(* PLC project , Arduino SRL Arduino PLC IDE Application 1.0.3.1 *)
(* stored: companyURL https://www.axelsoftware.it/, creationDateTime 2023-12-08T15:45:33 *)

VAR_GLOBAL  (* Global_vars *)
  cnt : INT;
  pickSeq : BOOL := FALSE;
  curSeq : INT := 10;
  auto : BOOL;
  manMode : BOOL;
  pickIndex : INT := 0;
  placePositionsY : ARRAY[0..3] OF INT := [7200, 10200, 13650, 16650];
  placeIndex : INT;
  placeSeq : BOOL;
  laserSeq : INT;
  pickPositionX : INT := 7975;
  placeClearZ : INT := 13600;
  workDone : BOOL := FALSE;
  pushSeq : BOOL;
  cutPositionsY : ARRAY[0..9] OF INT := [20970, 19000, 17030, 15060, 13090, 11120, 9150, 7180, 5210, 3240];
  cutBackX : INT := 15600;
  cutFrontX : INT := 18500;
  cutSeq : BOOL := FALSE;
  moveSpeed : INT := 375;
  min0 : INT := 0;
  min1 : INT := 0;
  hour0 : INT := 0;
  hour1 : INT := 0;
  placedCur : ARRAY[0..3] OF INT;
  timeReal : ARRAY[0..3] OF INT;
  timeRTC : ARRAY[0..3] OF INT;
  Solenoids AT %MX3.2 : ARRAY[0..3] OF BOOL;
  cutDigit : INT;
  engraveSeq : BOOL;
END_VAR

VAR_GLOBAL CONSTANT  (* Global_vars_Constant *)
  ZTop : INT := 14800;
  XOFF : INT := 0;
  YOFF : INT := 0;
  ZOFF : INT := 0;
  pickPositionsY : ARRAY[0..9] OF INT := [20900, 18930, 16960, 14990, 13020, 11050, 9080, 7100, 5140, 3600];
  pickClearanceZ : INT := 10000;
  placePositionX : INT := 19400;
  PBTimeOff : INT := 200;
  pushClearanceX : INT := 16350;
END_VAR

VAR_GLOBAL  (* I_O_mappings_DIO *)
  Sol1 AT %MX3.2 : BOOL;
  Sol2 AT %MX3.3 : BOOL;
  Sol3 AT %MX3.4 : BOOL;
  EnableXYZ AT %MX3.0 : BOOL;
  EnableA AT %MX3.1 : BOOL;
  Sol4 AT %MX3.5 : BOOL;
END_VAR

VAR_GLOBAL  (* I_O_mappings_DI *)
  XHome AT %IX0.0 : BOOL;
  YHome AT %IX0.1 : BOOL;
  ZHome AT %IX0.2 : BOOL;
END_VAR

VAR_GLOBAL  (* I_O_mappings_DO *)
  home2 : BOOL;
END_VAR

VAR_GLOBAL  (* I_O_mappings_AO *)
  laserPWM AT %QD1.1 : REAL;
END_VAR

PROGRAM TimeGetter

timeRTC[0] := minute MOD 10;
timeRTC[1] := minute / 10;

timeRTC[2] := hour MOD 10;
timeRTC[3] := hour / 10;

/* placedCur[3] is hour1 and also most significant.
If time changes, reset placedCur[x] to -1 and drop piece. */
IF(placedCur[3] = -1) THEN
	placeIndex := 3;

ELSIF(placedCur[2] = -1) THEN
	placeIndex := 2;

ELSIF(placedCur[1] = -1) THEN
	placeIndex := 1;
	
ELSIF(placedCur[0] = -1) THEN
	placeIndex := 0;

END_IF;

//set placedCur[x] to -1 when time changes, and not in motion.
END_PROGRAM

FUNCTION_BLOCK Engrave0
  VAR_INPUT
    YPOS0 : INT;
    XPOS0 : INT;
    XPOSACT : INT;
    YPOSACT : INT;
  END_VAR
  VAR_OUTPUT
    LASERPWM : REAL;
    XPOSOUT : INT;
    YPOSOUT : INT;
  END_VAR
  VAR_EXTERNAL
    curSeq : INT;
  END_VAR

IF (curSeq = 20) THEN
XPOSOUT := XPOS0 + 450;
YPOSOUT := YPOS0 + 450;
END_IF;


//Fire laser while moving through sequence
IF (curSeq > 20) AND (curSeq < 100) THEN
LASERPWM := 0.8;
ELSE
LASERPWM := 0.0;
END_IF;

IF (curSeq = 21) THEN
XPOSOUT := XPOS0 + 2505;
YPOSOUT := YPOS0 + 450;
END_IF;

IF (curSeq = 22) THEN
XPOSOUT := XPOS0 + 2505;
YPOSOUT := YPOS0 + 1520;
END_IF;

IF (curSeq = 23) THEN
XPOSOUT := XPOS0 + 450;
YPOSOUT := YPOS0 + 1520;
END_IF;

IF (curSeq = 24) THEN
XPOSOUT := XPOS0 + 450;
YPOSOUT := YPOS0 + 550;
END_IF;



//Move to next sequence if current sequence reaches its requested position.
//Might need another condition so CURSEQ doesn't keep incrementing
IF (XPOSOUT = XPOSACT) AND (YPOSOUT = YPOSACT) THEN 
curSeq := curSeq + 1;
END_IF;


//End of engrave sequence looking for 100
//23 is a placeholder for last sequence
IF(curSeq > 24) THEN
curSeq := 100;
LASERPWM := 0.0;

END_IF;
END_FUNCTION_BLOCK

FUNCTION_BLOCK Engrave1
  VAR_INPUT
    YPOS0 : INT;
    XPOS0 : INT;
    XPOSACT : INT;
    YPOSACT : INT;
  END_VAR
  VAR_OUTPUT
    LASERPWM : REAL;
    XPOSOUT : INT;
    YPOSOUT : INT;
  END_VAR
  VAR_EXTERNAL
    curSeq : INT;
  END_VAR

IF (curSeq = 20) THEN
XPOSOUT := XPOS0 + 768;
YPOSOUT := YPOS0 + 1303;
END_IF;


//Fire laser while moving through sequence
IF (curSeq > 20) AND (curSeq < 100) THEN
LASERPWM := 0.8;
ELSE
LASERPWM := 0.0;
END_IF;

IF (curSeq = 21) THEN
XPOSOUT := XPOS0 + 450;
YPOSOUT := YPOS0 + 985;
END_IF;

IF (curSeq = 22) THEN
XPOSOUT := XPOS0 + 2405;
YPOSOUT := YPOS0 + 985;
END_IF;

IF (curSeq = 23) THEN
XPOSOUT := XPOS0 + 2405;
YPOSOUT := YPOS0 + 1520;
END_IF;

IF (curSeq = 24) THEN
XPOSOUT := XPOS0 + 2505;
YPOSOUT := YPOS0 + 1520;
END_IF;

IF (curSeq = 25) THEN
XPOSOUT := XPOS0 + 2505;
YPOSOUT := YPOS0 + 450;
END_IF;



//Move to next sequence if current sequence reaches its requested position.
//Might need another condition so CURSEQ doesn't keep incrementing
IF (XPOSOUT = XPOSACT) AND (YPOSOUT = YPOSACT) THEN
curSeq := curSeq + 1;
END_IF;


//End of engrave sequence looking for 100
//23 is a placeholder for last sequence
IF(curSeq > 25) THEN
curSeq := 100;
LASERPWM := 0.0;
END_IF;
END_FUNCTION_BLOCK

FUNCTION_BLOCK Engrave2
  VAR_INPUT
    YPOS0 : INT;
    XPOS0 : INT;
    XPOSACT : INT;
    YPOSACT : INT;
  END_VAR
  VAR_OUTPUT
    LASERPWM : REAL;
    XPOSOUT : INT;
    YPOSOUT : INT;
  END_VAR
  VAR_EXTERNAL
    curSeq : INT;
  END_VAR

IF (curSeq = 20) THEN
XPOSOUT := XPOS0 + 900;
YPOSOUT := YPOS0 + 1520;
END_IF;


//Fire laser while moving through sequence
IF (curSeq > 20) AND (curSeq < 100) THEN
LASERPWM := 0.8;
ELSE
LASERPWM := 0.0;
END_IF;

IF (curSeq = 21) THEN
XPOSOUT := XPOS0 + 450;
YPOSOUT := YPOS0 + 1520;
END_IF;

IF (curSeq = 22) THEN
XPOSOUT := XPOS0 + 450;
YPOSOUT := YPOS0 + 450;
END_IF;

IF (curSeq = 23) THEN
XPOSOUT := XPOS0 + 1480;
YPOSOUT := YPOS0 + 450;
END_IF;

IF (curSeq = 24) THEN
XPOSOUT := XPOS0 + 1480;
YPOSOUT := YPOS0 + 1520;
END_IF;

IF (curSeq = 25) THEN
XPOSOUT := XPOS0 + 2505;
YPOSOUT := YPOS0 + 1520;
END_IF;

IF (curSeq = 26) THEN
XPOSOUT := XPOS0 + 2505;
YPOSOUT := YPOS0 + 450;
END_IF;



//Move to next sequence if current sequence reaches its requested position.
//Might need another condition so CURSEQ doesn't keep incrementing
IF (XPOSOUT = XPOSACT) AND (YPOSOUT = YPOSACT) THEN
curSeq := curSeq + 1;
END_IF;


//End of engrave sequence looking for 100
//23 is a placeholder for last sequence
IF(curSeq > 26) THEN
curSeq := 100;
LASERPWM := 0.0;
END_IF;
END_FUNCTION_BLOCK

FUNCTION_BLOCK Engrave3
  VAR_INPUT
    YPOS0 : INT;
    XPOS0 : INT;
    XPOSACT : INT;
    YPOSACT : INT;
  END_VAR
  VAR_OUTPUT
    LASERPWM : REAL;
    XPOSOUT : INT;
    YPOSOUT : INT;
  END_VAR
  VAR_EXTERNAL
    curSeq : INT;
  END_VAR

IF (curSeq = 20) THEN
XPOSOUT := XPOS0 + 450;
YPOSOUT := YPOS0 + 1520;
END_IF;


//Fire laser while moving through sequence
IF (curSeq > 20) AND (curSeq < 100) THEN
LASERPWM := 0.8;
ELSE
LASERPWM := 0.0;
END_IF;

IF (curSeq = 21) THEN
XPOSOUT := XPOS0 + 450;
YPOSOUT := YPOS0 + 450;
END_IF;

IF (curSeq = 22) THEN
XPOSOUT := XPOS0 + 1475;
YPOSOUT := YPOS0 + 450;
END_IF;

IF (curSeq = 23) THEN
XPOSOUT := XPOS0 + 1475;
YPOSOUT := YPOS0 + 1520;
END_IF;

IF (curSeq = 24) THEN
XPOSOUT := XPOS0 + 1575;
YPOSOUT := YPOS0 + 1520;
END_IF;

IF (curSeq = 25) THEN
XPOSOUT := XPOS0 + 1575;
YPOSOUT := YPOS0 + 450;
END_IF;

IF (curSeq = 26) THEN
XPOSOUT := XPOS0 + 2505;
YPOSOUT := YPOS0 + 450;
END_IF;

IF (curSeq = 27) THEN
XPOSOUT := XPOS0 + 2505;
YPOSOUT := YPOS0 + 1520;
END_IF;


//Move to next sequence if current sequence reaches its requested position.
//Might need another condition so CURSEQ doesn't keep incrementing
IF (XPOSOUT = XPOSACT) AND (YPOSOUT = YPOSACT) THEN
curSeq := curSeq + 1;
END_IF;


//End of engrave sequence looking for 100
//23 is a placeholder for last sequence
IF(curSeq > 27) THEN
curSeq := 100;
LASERPWM := 0.0;
END_IF;
END_FUNCTION_BLOCK

FUNCTION_BLOCK Engrave4
  VAR_INPUT
    YPOS0 : INT;
    XPOS0 : INT;
    XPOSACT : INT;
    YPOSACT : INT;
  END_VAR
  VAR_OUTPUT
    LASERPWM : REAL;
    XPOSOUT : INT;
    YPOSOUT : INT;
  END_VAR
  VAR_EXTERNAL
    curSeq : INT;
  END_VAR

IF (curSeq = 20) THEN
XPOSOUT := XPOS0 + 1412;
YPOSOUT := YPOS0 + 450;
END_IF;


//Fire laser while moving through sequence
IF (curSeq > 20) AND (curSeq < 100) THEN
LASERPWM := 0.8;
ELSE
LASERPWM := 0.0;
END_IF;

IF (curSeq = 21) THEN
XPOSOUT := XPOS0 + 1412;
YPOSOUT := YPOS0 + 1520;
END_IF;

IF (curSeq = 22) THEN
XPOSOUT := XPOS0 + 450;
YPOSOUT := YPOS0 + 741;
END_IF;

IF (curSeq = 23) THEN
XPOSOUT := XPOS0 + 2505;
YPOSOUT := YPOS0 + 741;
END_IF;



//Move to next sequence if current sequence reaches its requested position.
//Might need another condition so CURSEQ doesn't keep incrementing
IF (XPOSOUT = XPOSACT) AND (YPOSOUT = YPOSACT) THEN
curSeq := curSeq + 1;
END_IF;


//End of engrave sequence looking for 100
//23 is a placeholder for last sequence
IF(curSeq > 23) THEN
curSeq := 100;
LASERPWM := 0.0;
END_IF;
END_FUNCTION_BLOCK

FUNCTION_BLOCK Engrave5
  VAR_INPUT
    YPOS0 : INT;
    XPOS0 : INT;
    XPOSACT : INT;
    YPOSACT : INT;
  END_VAR
  VAR_OUTPUT
    LASERPWM : REAL;
    XPOSOUT : INT;
    YPOSOUT : INT;
  END_VAR
  VAR_EXTERNAL
    curSeq : INT;
  END_VAR

IF (curSeq = 20) THEN
XPOSOUT := XPOS0 + 450;
YPOSOUT := YPOS0 + 450;
END_IF;


//Fire laser while moving through sequence
IF (curSeq > 20) AND (curSeq < 100) THEN
LASERPWM := 0.8;
ELSE
LASERPWM := 0.0;
END_IF;

IF (curSeq = 21) THEN
XPOSOUT := XPOS0 + 450;
YPOSOUT := YPOS0 + 1520;
END_IF;

IF (curSeq = 22) THEN
XPOSOUT := XPOS0 + 1480;
YPOSOUT := YPOS0 + 1520;
END_IF;

IF (curSeq = 23) THEN
XPOSOUT := XPOS0 + 1480;
YPOSOUT := YPOS0 + 450;
END_IF;

IF (curSeq = 24) THEN
XPOSOUT := XPOS0 + 2505;
YPOSOUT := YPOS0 + 450;
END_IF;

IF (curSeq = 25) THEN
XPOSOUT := XPOS0 + 2505;
YPOSOUT := YPOS0 + 1520;
END_IF;



//Move to next sequence if current sequence reaches its requested position.
//Might need another condition so CURSEQ doesn't keep incrementing
IF (XPOSOUT = XPOSACT) AND (YPOSOUT = YPOSACT) THEN
curSeq := curSeq + 1;
END_IF;


//End of engrave sequence looking for 100
//23 is a placeholder for last sequence
IF(curSeq > 25) THEN
curSeq := 100;
LASERPWM := 0.0;
END_IF;
END_FUNCTION_BLOCK

FUNCTION_BLOCK Engrave6
  VAR_INPUT
    YPOS0 : INT;
    XPOS0 : INT;
    XPOSACT : INT;
    YPOSACT : INT;
  END_VAR
  VAR_OUTPUT
    LASERPWM : REAL;
    XPOSOUT : INT;
    YPOSOUT : INT;
  END_VAR
  VAR_EXTERNAL
    curSeq : INT;
  END_VAR

IF (curSeq = 20) THEN
XPOSOUT := XPOS0 + 450;
YPOSOUT := YPOS0 + 450;
END_IF;


//Fire laser while moving through sequence
IF (curSeq > 20) AND (curSeq < 100) THEN
LASERPWM := 0.8;
ELSE
LASERPWM := 0.0;
END_IF;

IF (curSeq = 21) THEN
XPOSOUT := XPOS0 + 450;
YPOSOUT := YPOS0 + 1520;
END_IF;

IF (curSeq = 22) THEN
XPOSOUT := XPOS0 + 1475;
YPOSOUT := YPOS0 + 1520;
END_IF;

IF (curSeq = 23) THEN
XPOSOUT := XPOS0 + 1475;
YPOSOUT := YPOS0 + 450;
END_IF;

IF (curSeq = 24) THEN
XPOSOUT := XPOS0 + 2505;
YPOSOUT := YPOS0 + 450;
END_IF;

IF (curSeq = 25) THEN
XPOSOUT := XPOS0 + 2505;
YPOSOUT := YPOS0 + 1520;
END_IF;

IF (curSeq = 26) THEN
XPOSOUT := XPOS0 + 1575;
YPOSOUT := YPOS0 + 1520;
END_IF;


//Move to next sequence if current sequence reaches its requested position.
//Might need another condition so CURSEQ doesn't keep incrementing
IF (XPOSOUT = XPOSACT) AND (YPOSOUT = YPOSACT) THEN
curSeq := curSeq + 1;
END_IF;


//End of engrave sequence looking for 100
IF(curSeq > 26) THEN
curSeq := 100;
LASERPWM := 0.0;
END_IF;
END_FUNCTION_BLOCK

FUNCTION_BLOCK Engrave7
  VAR_INPUT
    YPOS0 : INT;
    XPOS0 : INT;
    XPOSACT : INT;
    YPOSACT : INT;
  END_VAR
  VAR_OUTPUT
    LASERPWM : REAL;
    XPOSOUT : INT;
    YPOSOUT : INT;
  END_VAR
  VAR_EXTERNAL
    curSeq : INT;
  END_VAR

IF (curSeq = 20) THEN
XPOSOUT := XPOS0 + 450;
YPOSOUT := YPOS0 + 1520;
END_IF;


//Fire laser while moving through sequence
IF (curSeq > 20) AND (curSeq < 100) THEN
LASERPWM := 0.8;
ELSE
LASERPWM := 0.0;
END_IF;

IF (curSeq = 21) THEN
XPOSOUT := XPOS0 + 450;
YPOSOUT := YPOS0 + 450;
END_IF;

IF (curSeq = 22) THEN
XPOSOUT := XPOS0 + 2505;
YPOSOUT := YPOS0 + 1520;
END_IF;



//Move to next sequence if current sequence reaches its requested position.
//Might need another condition so CURSEQ doesn't keep incrementing
IF (XPOSOUT = XPOSACT) AND (YPOSOUT = YPOSACT) THEN
curSeq := curSeq + 1;
END_IF;


//End of engrave sequence looking for 100
IF(curSeq > 22) THEN
curSeq := 100;
LASERPWM := 0.0;
END_IF;
END_FUNCTION_BLOCK

FUNCTION_BLOCK Engrave8
  VAR_INPUT
    YPOS0 : INT;
    XPOS0 : INT;
    XPOSACT : INT;
    YPOSACT : INT;
  END_VAR
  VAR_OUTPUT
    LASERPWM : REAL;
    XPOSOUT : INT;
    YPOSOUT : INT;
  END_VAR
  VAR_EXTERNAL
    curSeq : INT;
  END_VAR

IF (curSeq = 20) THEN
XPOSOUT := XPOS0 + 450;
YPOSOUT := YPOS0 + 450;
END_IF;


//Fire laser while moving through sequence
IF (curSeq > 20) AND (curSeq < 100) THEN
LASERPWM := 0.8;
ELSE
LASERPWM := 0.0;
END_IF;

IF (curSeq = 21) THEN
XPOSOUT := XPOS0 + 450;
YPOSOUT := YPOS0 + 1520;
END_IF;

IF (curSeq = 22) THEN
XPOSOUT := XPOS0 + 1430;
YPOSOUT := YPOS0 + 1520;
END_IF;

IF (curSeq = 22) THEN
XPOSOUT := XPOS0 + 1430;
YPOSOUT := YPOS0 + 550;
END_IF;

IF (curSeq = 23) THEN
XPOSOUT := XPOS0 + 1530;
YPOSOUT := YPOS0 + 550;
END_IF;

IF (curSeq = 24) THEN
XPOSOUT := XPOS0 + 1530;
YPOSOUT := YPOS0 + 1520;
END_IF;

IF (curSeq = 25) THEN
XPOSOUT := XPOS0 + 2505;
YPOSOUT := YPOS0 + 1520;
END_IF;

IF (curSeq = 26) THEN
XPOSOUT := XPOS0 + 2505;
YPOSOUT := YPOS0 + 450;
END_IF;

IF (curSeq = 27) THEN
XPOSOUT := XPOS0 + 550;
YPOSOUT := YPOS0 + 450;
END_IF;


//Move to next sequence if current sequence reaches its requested position.
//Might need another condition so CURSEQ doesn't keep incrementing
IF (XPOSOUT = XPOSACT) AND (YPOSOUT = YPOSACT) THEN
curSeq := curSeq + 1;
END_IF;


//End of engrave sequence looking for 100
IF(curSeq > 27) THEN
curSeq := 100;
LASERPWM := 0.0;
END_IF;
END_FUNCTION_BLOCK

FUNCTION_BLOCK Engrave9
  VAR_INPUT
    YPOS0 : INT;
    XPOS0 : INT;
    XPOSACT : INT;
    YPOSACT : INT;
  END_VAR
  VAR_OUTPUT
    LASERPWM : REAL;
    XPOSOUT : INT;
    YPOSOUT : INT;
  END_VAR
  VAR_EXTERNAL
    curSeq : INT;
  END_VAR

IF (curSeq = 20) THEN
XPOSOUT := XPOS0 + 1475;
YPOSOUT := YPOS0 + 550;
END_IF;


//Fire laser while moving through sequence
IF (curSeq > 20) AND (curSeq < 100) THEN
LASERPWM := 0.8;
ELSE
LASERPWM := 0.0;
END_IF;

IF (curSeq = 21) THEN
XPOSOUT := XPOS0 + 1475;
YPOSOUT := YPOS0 + 1520;
END_IF;

IF (curSeq = 22) THEN
XPOSOUT := XPOS0 + 450;
YPOSOUT := YPOS0 + 1520;
END_IF;

IF (curSeq = 22) THEN
XPOSOUT := XPOS0 + 450;
YPOSOUT := YPOS0 + 450;
END_IF;

IF (curSeq = 23) THEN
XPOSOUT := XPOS0 + 2505;
YPOSOUT := YPOS0 + 450;
END_IF;

IF (curSeq = 24) THEN
XPOSOUT := XPOS0 + 2505;
YPOSOUT := YPOS0 + 1520;
END_IF;



//Move to next sequence if current sequence reaches its requested position.
//Might need another condition so CURSEQ doesn't keep incrementing
IF (XPOSOUT = XPOSACT) AND (YPOSOUT = YPOSACT) THEN
curSeq := curSeq + 1;
END_IF;


//End of engrave sequence looking for 100
IF(curSeq > 24) THEN
curSeq := 100;
LASERPWM := 0.0;
END_IF;
END_FUNCTION_BLOCK

CONFIGURATION Configuration
  RESOURCE Resource ON PLC
    VAR_GLOBAL  (* Global_vars *)
      cnt : INT;
      pickSeq : BOOL := FALSE;
      curSeq : INT := 10;
      auto : BOOL;
      manMode : BOOL;
      pickIndex : INT := 0;
      placePositionsY : ARRAY[0..3] OF INT := [7200, 10200, 13650, 16650];
      placeIndex : INT;
      placeSeq : BOOL;
      laserSeq : INT;
      pickPositionX : INT := 7975;
      placeClearZ : INT := 13600;
      workDone : BOOL := FALSE;
      pushSeq : BOOL;
      cutPositionsY : ARRAY[0..9] OF INT := [20970, 19000, 17030, 15060, 13090, 11120, 9150, 7180, 5210, 3240];
      cutBackX : INT := 15600;
      cutFrontX : INT := 18500;
      cutSeq : BOOL := FALSE;
      moveSpeed : INT := 375;
      min0 : INT := 0;
      min1 : INT := 0;
      hour0 : INT := 0;
      hour1 : INT := 0;
      placedCur : ARRAY[0..3] OF INT;
      timeReal : ARRAY[0..3] OF INT;
      timeRTC : ARRAY[0..3] OF INT;
      Solenoids AT %MX3.2 : ARRAY[0..3] OF BOOL;
      cutDigit : INT;
      engraveSeq : BOOL;
    END_VAR
    VAR_GLOBAL CONSTANT  (* Global_vars_Constant *)
      ZTop : INT := 14800;
      XOFF : INT := 0;
      YOFF : INT := 0;
      ZOFF : INT := 0;
      pickPositionsY : ARRAY[0..9] OF INT := [20900, 18930, 16960, 14990, 13020, 11050, 9080, 7100, 5140, 3600];
      pickClearanceZ : INT := 10000;
      placePositionX : INT := 19400;
      PBTimeOff : INT := 200;
      pushClearanceX : INT := 16350;
    END_VAR
    VAR_GLOBAL  (* I_O_mappings_DIO *)
      Sol1 AT %MX3.2 : BOOL;
      Sol2 AT %MX3.3 : BOOL;
      Sol3 AT %MX3.4 : BOOL;
      EnableXYZ AT %MX3.0 : BOOL;
      EnableA AT %MX3.1 : BOOL;
      Sol4 AT %MX3.5 : BOOL;
    END_VAR
    VAR_GLOBAL  (* I_O_mappings_DI *)
      XHome AT %IX0.0 : BOOL;
      YHome AT %IX0.1 : BOOL;
      ZHome AT %IX0.2 : BOOL;
    END_VAR
    VAR_GLOBAL  (* I_O_mappings_DO *)
      home2 : BOOL;
    END_VAR
    VAR_GLOBAL  (* I_O_mappings_AO *)
      laserPWM AT %QD1.1 : REAL;
    END_VAR
  END_RESOURCE
END_CONFIGURATION
